PROGRAM Nappivalot
VAR
first_cycle : BOOL := TRUE;
nappilasku : INT;
END_VAR

IF io.out_punainenvalo AND io.in_nappi_punainen THEN
	io.out_punainenvalo:=FALSE; 
	io.out_sininenvalo:=TRUE;
END_IF

IF io.out_sininenvalo AND io.in_nappi_sininen THEN
	io.out_sininenvalo:=FALSE;
	io.out_valkoinenvalo:=TRUE;
END_IF

IF io.out_valkoinenvalo AND io.in_nappi_valkoinen THEN
	io.out_valkoinenvalo:=FALSE;
	io.out_punainenvalo:=TRUE;
END_IF



IF first_cycle THEN
	io.out_punainenvalo:=TRUE;
	first_cycle:=FALSE;
END_IF

END_PROGRAM

(* stored: Version 1.1.0.1, ProductVersion 3.1.4024.10
   POU Nappivalot: Id {869e099f-69a8-43b1-a3d1-a06029cff49e}, SpecialFunc None *)
